// TIA Portal V19 export
DATA_BLOCK "DB_System"   // DB3
{ S7_Optimized_Access := 'TRUE' }
// stored: AutoNumber false, MemoryReserve 100
   VAR
      datetime : Struct
         current : DTL := DTL#2025-09-17-14:58:30.265837800;
      END_STRUCT;
      firstCycle : Bool := TRUE;
      reqPointers : Bool := FALSE;
      reqParametrizations : Bool := FALSE;
   END_VAR
   VAR RETAIN
      modulesGroup : Struct
         ADIN { S7_SetPoint := 'True'} : Bool := FALSE;
         AIN { S7_SetPoint := 'True'} : Bool := TRUE;
         DIFF { S7_SetPoint := 'True'} : Bool := FALSE;
         DIN { S7_SetPoint := 'True'} : Bool := TRUE;
         MTR { S7_SetPoint := 'True'} : Bool := TRUE;
         MTRDIR { S7_SetPoint := 'True'} : Bool := TRUE;
         MTRLIN { S7_SetPoint := 'True'} : Bool := FALSE;
         VLV { S7_SetPoint := 'True'} : Bool := FALSE;
         CVLV { S7_SetPoint := 'True'} : Bool := FALSE;
      END_STRUCT;
   END_VAR
   VAR
      reqQuickSetup { S7_SetPoint := 'True'} : "modTypes";
   END_VAR
BEGIN
   reqQuickSetup.adin := FALSE;
   reqQuickSetup.ain := FALSE;
   reqQuickSetup.cvlv := FALSE;
   reqQuickSetup.din := FALSE;
   reqQuickSetup.mtr := FALSE;
   reqQuickSetup.mtrDir := FALSE;
   reqQuickSetup.mtrLin := FALSE;
   reqQuickSetup.vlv := FALSE;
END_DATA_BLOCK
